FUNCTION_BLOCK CONSTRUCT_DDS_ID (* Function Block to Construct DDS COM ID *)
  (* Standard: 61499-2 *)
  (* Version 1.0, 2023-03-08, Tim Hesse *)
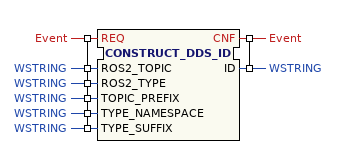
  EVENT_INPUT
    REQ WITH ROS2_TOPIC, ROS2_TYPE, TOPIC_PREFIX, TYPE_NAMESPACE, TYPE_SUFFIX; (* Service Request *)
  END_EVENT
  EVENT_OUTPUT
    CNF WITH ID; (* Confirmation of Requested Service *)
  END_EVENT
  VAR_INPUT
    ROS2_TOPIC : WSTRING; (* Topic Name from ROS 2 *)
    ROS2_TYPE : WSTRING; (* Type Name from ROS 2 *)
    TOPIC_PREFIX : WSTRING; (* Prefix for DDS Topic *)
    TYPE_NAMESPACE : WSTRING; (* Namespace for DDS Type *)
    TYPE_SUFFIX : WSTRING; (* Suffix for DDS Type *)
  END_VAR
  VAR_OUTPUT
    ID : WSTRING; (* Service Status *)
  END_VAR
  SERVICE APPLICATION/RESOURCE (* Function Block to Construct DDS COM ID *)
    SEQUENCE normal_establishment
      APPLICATION.INIT+(PARAMS) -> RESOURCE.initialize(PARAMS) -> APPLICATION.INITO+();
    END_SEQUENCE
    SEQUENCE unsuccessful_establishment
      APPLICATION.INIT+(PARAMS) -> RESOURCE.initialize(PARAMS) -> APPLICATION.INITO-(STATUS);
    END_SEQUENCE
    SEQUENCE request_confirm
      APPLICATION.REQ+(SD) -> RESOURCE.request(SD) -> APPLICATION.CNF+(RD);
    END_SEQUENCE
    SEQUENCE request_inhibited
      APPLICATION.REQ-(SD) -> APPLICATION.CNF-(STATUS);
    END_SEQUENCE
    SEQUENCE request_error
      APPLICATION.REQ+(SD) -> RESOURCE.request(SD) -> APPLICATION.CNF-(STATUS);
    END_SEQUENCE
    SEQUENCE indication_response
      RESOURCE.indicate(RD) -> APPLICATION.IND+(RD);
      APPLICATION.RSP(QI,SD) -> RESOURCE.response(QI,SD);
    END_SEQUENCE
    SEQUENCE indication_inhibited
      RESOURCE.indicate(RD,QI=FALSE) -> RESOURCE.inhibited();
    END_SEQUENCE
    SEQUENCE error_indication
      RESOURCE.error(STATUS) -> APPLICATION.IND-(STATUS);
    END_SEQUENCE
    SEQUENCE application_initiated_termination
      APPLICATION.INIT-() -> RESOURCE.terminate() -> APPLICATION.INITO-(STATUS);
    END_SEQUENCE
    SEQUENCE resource_initiated_termination
      -> APPLICATION.INITO-(STATUS);
    END_SEQUENCE
  END_SERVICE
END_FUNCTION_BLOCK
